PROGRAM SafetyInterface_MtrCntrl051
VAR
	
	pMtrRunning: POINTER TO ConvMtrRunningPuck;
	pSafety: POINTER TO Plc2PlcDataSafetyPuckConv;
	
// Stn051_05_StnMain.MotorCtrl
// Call to motor control function block for each main line motor	
// Blue Return - Enc52:  5,6  Enc53: 3,4,5,6
// Red Return  - Enc52:  3,4   Enc53:2
// Grn Return  - Enc52: 1,2   Enc53: 1
//  Blu receive bypass - Enc52: 7
	{attribute 'TcLinkToOSO':= '	
		.Enc052Mtr01.iDisconnectOk :=  <0,1,3>TIIB[N16S00 (AL1332)]^N16S03 (AL2341)^TxPDO^input byte 3;
		.Enc052Mtr02.iDisconnectOk :=  <0,1,3>TIIB[N16S00 (AL1332)]^N16S07 (AL2341)^TxPDO^input byte 1;
		.Enc052Mtr03.iDisconnectOk :=  <0,1,4>TIIB[N16S00 (AL1332)]^N16S03 (AL2341)^TxPDO^input byte 1;
		.Enc052Mtr04.iDisconnectOk :=  <0,1,3>TIIB[N16S00 (AL1332)]^N16S07 (AL2341)^TxPDO^input byte 3;
		.Enc052Mtr05.iDisconnectOk :=  <0,1,4>TIIB[N16S00 (AL1332)]^N16S03 (AL2341)^TxPDO^input byte 3;
		.Enc052Mtr06.iDisconnectOk :=  <0,1,4>TIIB[N16S00 (AL1332)]^N16S07 (AL2341)^TxPDO^input byte 1;
		.Enc052Mtr07.iDisconnectOk :=  <0,1,4>TIIB[N16S00 (AL1332)]^N16S07 (AL2341)^TxPDO^input byte 3;
		.Enc053Mtr01.iDisconnectOk :=  <0,1,2>TIIB[N21S00 (AL1332)]^N21S01 (AL2341)^TxPDO^input byte 3;
		.Enc053Mtr02.iDisconnectOk :=  <0,1,3>TIIB[N21S00 (AL1332)]^N21S01 (AL2341)^TxPDO^input byte 1;
		.Enc053Mtr03.iDisconnectOk :=  <0,1,3>TIIB[N21S00 (AL1332)]^N21S01 (AL2341)^TxPDO^input byte 1;
		.Enc053Mtr04.iDisconnectOk :=  <0,1,3>TIIB[N21S00 (AL1332)]^N21S01 (AL2341)^TxPDO^input byte 1;
		.Enc053Mtr05.iDisconnectOk :=  <0,1,4>TIIB[N24S00 (AL1332)]^N24S05 (AL2341)^TxPDO^input byte 3;
		.Enc053Mtr06.iDisconnectOk :=  <0,1,3>TIIB[N21S00 (AL1332)]^N21S01 (AL2341)^TxPDO^input byte 1'}
	{attribute 'TcLinkTo':= '	
		.Enc052Mtr01.iOverloadTripped := TIIB[N15S06 (EL1008)]^Channel 6^Input;
		.Enc052Mtr02.iOverloadTripped := TIIB[N15S06 (EL1008)]^Channel 8^Input;
		.Enc052Mtr03.iOverloadTripped := TIIB[N15S07 (EL1008)]^Channel 2^Input;
		.Enc052Mtr04.iOverloadTripped := TIIB[N15S07 (EL1008)]^Channel 4^Input;
		.Enc052Mtr05.iOverloadTripped := TIIB[N15S07 (EL1008)]^Channel 6^Input;
		.Enc052Mtr06.iOverloadTripped := TIIB[N15S07 (EL1008)]^Channel 8^Input;
		.Enc052Mtr07.iOverloadTripped := TIIB[N15S08 (EL1008)]^Channel 2^Input;
		.Enc053Mtr01.iOverloadTripped := TIIB[N20S06 (EL1008)]^Channel 6^Input;
		.Enc053Mtr02.iOverloadTripped := TIIB[N20S06 (EL1008)]^Channel 8^Input;
		.Enc053Mtr03.iOverloadTripped := TIIB[N20S07 (EL1008)]^Channel 2^Input;
		.Enc053Mtr04.iOverloadTripped := TIIB[N20S07 (EL1008)]^Channel 4^Input;
		.Enc053Mtr05.iOverloadTripped := TIIB[N20S07 (EL1008)]^Channel 6^Input;
		.Enc053Mtr06.iOverloadTripped := TIIB[N20S07 (EL1008)]^Channel 8^Input;
		.Enc052Mtr01.iRunning := TIIB[N15S06 (EL1008)]^Channel 5^Input;
		.Enc052Mtr02.iRunning := TIIB[N15S06 (EL1008)]^Channel 7^Input;
		.Enc052Mtr03.iRunning := TIIB[N15S07 (EL1008)]^Channel 1^Input;
		.Enc052Mtr04.iRunning := TIIB[N15S07 (EL1008)]^Channel 3^Input;
		.Enc052Mtr05.iRunning := TIIB[N15S07 (EL1008)]^Channel 5^Input;
		.Enc052Mtr06.iRunning := TIIB[N15S07 (EL1008)]^Channel 7^Input;
		.Enc052Mtr07.iRunning := TIIB[N15S08 (EL1008)]^Channel 1^Input;
		.Enc053Mtr01.iRunning := TIIB[N20S06 (EL1008)]^Channel 5^Input;
		.Enc053Mtr02.iRunning := TIIB[N20S06 (EL1008)]^Channel 7^Input;
		.Enc053Mtr03.iRunning := TIIB[N20S07 (EL1008)]^Channel 1^Input;
		.Enc053Mtr04.iRunning := TIIB[N20S07 (EL1008)]^Channel 3^Input;
		.Enc053Mtr05.iRunning := TIIB[N20S07 (EL1008)]^Channel 5^Input;
		.Enc053Mtr06.iRunning := TIIB[N20S07 (EL1008)]^Channel 7^Input;
		.Enc052Mtr01.oRun := TIIB[N15S12 (EL2008)]^Channel 5^Output;
		.Enc052Mtr02.oRun := TIIB[N15S12 (EL2008)]^Channel 6^Output;
		.Enc052Mtr03.oRun := TIIB[N15S12 (EL2008)]^Channel 7^Output;
		.Enc052Mtr04.oRun := TIIB[N15S12 (EL2008)]^Channel 8^Output;
		.Enc052Mtr05.oRun := TIIB[N15S13 (EL2008)]^Channel 1^Output;
		.Enc052Mtr06.oRun := TIIB[N15S13 (EL2008)]^Channel 2^Output;
		.Enc052Mtr07.oRun := TIIB[N15S13 (EL2008)]^Channel 3^Output;
		.Enc053Mtr01.oRun := TIIB[N20S12 (EL2008)]^Channel 4^Output;
		.Enc053Mtr02.oRun := TIIB[N20S12 (EL2008)]^Channel 5^Output;
		.Enc053Mtr03.oRun := TIIB[N20S12 (EL2008)]^Channel 6^Output;
		.Enc053Mtr04.oRun := TIIB[N20S12 (EL2008)]^Channel 7^Output;
		.Enc053Mtr05.oRun := TIIB[N20S12 (EL2008)]^Channel 8^Output;
		.Enc053Mtr06.oRun := TIIB[N20S13 (EL2008)]^Channel 1^Output'}
	MtrCtrls: ConvMtrCtrlsPuck;

	MtrNOKtoRun : BOOL;	  	//not used at this time, see the attached action for details.
	cntMotorStartIndex: DINT;	
	tmrMotorStartIndex: TON;


END_VAR
VAR CONSTANT	
	
	cMaxMotorStartIndex :DINT := 9;  //If starting pairs of motors  adjust to max number of motors "per enclosure" /2
	
END_VAR

pMtrRunning := ADR(gProduced_SafetyInterfaceConv.MtrRunning);
pSafety := ADR(gProduced_SafetyInterfaceConv);

//Create sequenced motor start index - to prevent inrush overloads at time of motor start		
tmrMotorStartIndex(IN:=NOT tmrMotorStartIndex.Q,PT:=T#300ms);		
IF tmrMotorStartIndex.Q THEN 		
	cntMotorStartIndex := cntMotorStartIndex + 1;	
	IF cntMotorStartIndex > cMaxMotorStartIndex THEN 	
		cntMotorStartIndex := 1;
	END_IF	
END_IF		

// Call action code block that does call for each main line motor		
MotorCtrl();

//distibute the incoming stn data (consumed data from stn) to single produced outgoing to all stns
//MEMCPY(ADR(gProduced_SafetyInterfaceConv.gMtrRunningStn051), ADR(gMtrRunning), SizeOf(gProduced_SafetyInterfaceConv.gMtrRunningStn051));

ACTION MotorCtrl:
// Stn051_05_StnMain.MotorCtrl
// Call to motor control function block for each main line motor	
// Blue Return - Enc52:  5,6  Enc53: 3,4,5,6
// Red Return  - Enc52:  3,4   Enc53:2
// Grn Return  - Enc52: 1,2   Enc53: 1
//  Blu receive bypass - Enc52: 7

MtrCtrls.Enc052Mtr01(	
	CycleAuto := gConsumed_Stn051ToSafetyInterface.CycleAuto,
	CycleReset := gConsumed_Stn051ToSafetyInterface.CycleReset,
	NOKtoRun := pSafety^.Enc052.iEstopRlyTripped,	
//	NOKtoRun := pSafety^.Enc052.iEstopRlyTripped OR 
//		NOT gConsumed_Stn051ToSafetyInterface.Stn051PLCData[2].3 OR 
//		NOT gConsumed_Stn051ToSafetyInterface_OK,		
	StartIndexThisMotor := 1,
	StartIndexCurrent := cntMotorStartIndex,
	hoMtrName := 'Enc052-Mtr1',
	MtrRunning => pMtrRunning^.Enc052Mtr01);

MtrCtrls.Enc052Mtr02(	
	CycleAuto := gConsumed_Stn051ToSafetyInterface.CycleAuto,
	CycleReset := gConsumed_Stn051ToSafetyInterface.CycleReset,
	NOKtoRun := pSafety^.Enc052.iEstopRlyTripped,	
//	NOKtoRun := pSafety^.Enc052.iEstopRlyTripped OR 
//		NOT gConsumed_Stn051ToSafetyInterface.Stn051PLCData[2].3 OR 
//		NOT gConsumed_Stn051ToSafetyInterface_OK,		
	StartIndexThisMotor := 1,
	StartIndexCurrent := cntMotorStartIndex,
	hoMtrName := 'Enc052-Mtr2',
	MtrRunning => pMtrRunning^.Enc052Mtr02);

MtrCtrls.Enc052Mtr03(	
	CycleAuto := gConsumed_Stn051ToSafetyInterface.CycleAuto,
	CycleReset := gConsumed_Stn051ToSafetyInterface.CycleReset,
	NOKtoRun := pSafety^.Enc052.iEstopRlyTripped,	
//	NOKtoRun := pSafety^.Enc052.iEstopRlyTripped OR 
//		NOT gConsumed_Stn051ToSafetyInterface.Stn051PLCData[2].3 OR 
//		NOT gConsumed_Stn051ToSafetyInterface_OK,		
	StartIndexThisMotor := 2,
	StartIndexCurrent := cntMotorStartIndex,
	hoMtrName := 'Enc052-Mtr3',
	MtrRunning => pMtrRunning^.Enc052Mtr03);

MtrCtrls.Enc052Mtr04(	
	CycleAuto := gConsumed_Stn051ToSafetyInterface.CycleAuto,
	CycleReset := gConsumed_Stn051ToSafetyInterface.CycleReset,
	NOKtoRun := pSafety^.Enc052.iEstopRlyTripped,	
//	NOKtoRun := pSafety^.Enc052.iEstopRlyTripped OR 
//		NOT gConsumed_Stn051ToSafetyInterface.Stn051PLCData[2].3 OR 
//		NOT gConsumed_Stn051ToSafetyInterface_OK,		
	StartIndexThisMotor := 2,
	StartIndexCurrent := cntMotorStartIndex,
	hoMtrName := 'Enc052-Mtr4',
	MtrRunning => pMtrRunning^.Enc052Mtr04);

MtrCtrls.Enc052Mtr05(	
	CycleAuto := gConsumed_Stn051ToSafetyInterface.CycleAuto,
	CycleReset := gConsumed_Stn051ToSafetyInterface.CycleReset,
	NOKtoRun := pSafety^.Enc052.iEstopRlyTripped,	
//	NOKtoRun := pSafety^.Enc052.iEstopRlyTripped OR 
//		NOT gConsumed_Stn051ToSafetyInterface.Stn051PLCData[2].3 OR 
//		NOT gConsumed_Stn051ToSafetyInterface_OK,		
	StartIndexThisMotor := 3,
	StartIndexCurrent := cntMotorStartIndex,
	hoMtrName := 'Enc052-Mtr5',
	MtrRunning => pMtrRunning^.Enc052Mtr05);

MtrCtrls.Enc052Mtr06(	
	CycleAuto := gConsumed_Stn051ToSafetyInterface.CycleAuto,
	CycleReset := gConsumed_Stn051ToSafetyInterface.CycleReset,
	NOKtoRun := pSafety^.Enc052.iEstopRlyTripped,	
//	NOKtoRun := pSafety^.Enc052.iEstopRlyTripped OR 
//		NOT gConsumed_Stn051ToSafetyInterface.Stn051PLCData[2].3 OR 
//		NOT gConsumed_Stn051ToSafetyInterface_OK,		
	StartIndexThisMotor := 3,
	StartIndexCurrent := cntMotorStartIndex,
	hoMtrName := 'Enc052-Mtr6',
	MtrRunning => pMtrRunning^.Enc052Mtr06);

MtrCtrls.Enc052Mtr07(	
	CycleAuto := gConsumed_Stn051ToSafetyInterface.CycleAuto,
	CycleReset := gConsumed_Stn051ToSafetyInterface.CycleReset,
	NOKtoRun := pSafety^.Enc052.iEstopRlyTripped,	
//	NOKtoRun := pSafety^.Enc052.iEstopRlyTripped OR 
//		NOT gConsumed_Stn051ToSafetyInterface.Stn051PLCData[2].3 OR 
//		NOT gConsumed_Stn051ToSafetyInterface_OK,		
	StartIndexThisMotor := 4,
	StartIndexCurrent := cntMotorStartIndex,
	hoMtrName := 'Enc052-Mtr7',
	MtrRunning => pMtrRunning^.Enc052Mtr07);

MtrCtrls.Enc053Mtr01(	
	CycleAuto := gConsumed_Stn051ToSafetyInterface.CycleAuto,
	CycleReset := gConsumed_Stn051ToSafetyInterface.CycleReset,
	NOKtoRun := pSafety^.Enc053.iEstopRlyTripped,	
//	NOKtoRun := pSafety^.Enc053.iEstopRlyTripped OR 
//		NOT gConsumed_Stn051ToSafetyInterface.Stn051PLCData[2].3 OR 
//		NOT gConsumed_Stn051ToSafetyInterface_OK,		
	StartIndexThisMotor := 1,
	StartIndexCurrent := cntMotorStartIndex,
	hoMtrName := 'Enc053-Mtr1',
	MtrRunning => pMtrRunning^.Enc053Mtr01);

MtrCtrls.Enc053Mtr02(	
	CycleAuto := gConsumed_Stn051ToSafetyInterface.CycleAuto,
	CycleReset := gConsumed_Stn051ToSafetyInterface.CycleReset,
	NOKtoRun := pSafety^.Enc053.iEstopRlyTripped,	
//	NOKtoRun := pSafety^.Enc053.iEstopRlyTripped OR 
//		NOT gConsumed_Stn051ToSafetyInterface.Stn051PLCData[2].3 OR 
//		NOT gConsumed_Stn051ToSafetyInterface_OK,		
	StartIndexThisMotor := 1,
	StartIndexCurrent := cntMotorStartIndex,
	hoMtrName := 'Enc053-Mtr2',
	MtrRunning => pMtrRunning^.Enc053Mtr02);

MtrCtrls.Enc053Mtr03(	
	CycleAuto := gConsumed_Stn051ToSafetyInterface.CycleAuto,
	CycleReset := gConsumed_Stn051ToSafetyInterface.CycleReset,
	NOKtoRun := pSafety^.Enc053.iEstopRlyTripped,	
//	NOKtoRun := pSafety^.Enc053.iEstopRlyTripped OR 
//		NOT gConsumed_Stn051ToSafetyInterface.Stn051PLCData[2].3 OR 
//		NOT gConsumed_Stn051ToSafetyInterface_OK,		
	StartIndexThisMotor := 2,
	StartIndexCurrent := cntMotorStartIndex,
	hoMtrName := 'Enc053-Mtr3',
	MtrRunning => pMtrRunning^.Enc053Mtr03);

MtrCtrls.Enc053Mtr04(	
	CycleAuto := gConsumed_Stn051ToSafetyInterface.CycleAuto,
	CycleReset := gConsumed_Stn051ToSafetyInterface.CycleReset,
	NOKtoRun := pSafety^.Enc053.iEstopRlyTripped,	
//	NOKtoRun := pSafety^.Enc053.iEstopRlyTripped OR 
//		NOT gConsumed_Stn051ToSafetyInterface.Stn051PLCData[2].3 OR 
//		NOT gConsumed_Stn051ToSafetyInterface_OK,		
	StartIndexThisMotor := 2,
	StartIndexCurrent := cntMotorStartIndex,
	hoMtrName := 'Enc053-Mtr4',
	MtrRunning => pMtrRunning^.Enc053Mtr04);

MtrCtrls.Enc053Mtr05(	
	CycleAuto := gConsumed_Stn051ToSafetyInterface.CycleAuto,
	CycleReset := gConsumed_Stn051ToSafetyInterface.CycleReset,
	NOKtoRun := pSafety^.Enc053.iEstopRlyTripped,	
//	NOKtoRun := pSafety^.Enc053.iEstopRlyTripped OR 
//		NOT gConsumed_Stn051ToSafetyInterface.Stn051PLCData[2].3 OR 
//		NOT gConsumed_Stn051ToSafetyInterface_OK,		
	StartIndexThisMotor := 3,
	StartIndexCurrent := cntMotorStartIndex,
	hoMtrName := 'Enc053-Mtr5',
	MtrRunning => pMtrRunning^.Enc053Mtr05);

MtrCtrls.Enc053Mtr06(	
	CycleAuto := gConsumed_Stn051ToSafetyInterface.CycleAuto,
	CycleReset := gConsumed_Stn051ToSafetyInterface.CycleReset,
	NOKtoRun := pSafety^.Enc053.iEstopRlyTripped,	
//	NOKtoRun := pSafety^.Enc053.iEstopRlyTripped OR 
//		NOT gConsumed_Stn051ToSafetyInterface.Stn051PLCData[2].3 OR 
//		NOT gConsumed_Stn051ToSafetyInterface_OK,		
	StartIndexThisMotor := 3,
	StartIndexCurrent := cntMotorStartIndex,
	hoMtrName := 'Enc053-Mtr6',
	MtrRunning => pMtrRunning^.Enc053Mtr06);
	
//For each motor that the station needs running information but NOT actually controlling the output… 
//(populate the running bit from the produced consumed logic)

// Populate motor running for motors controlled (outputs linked) by other stations
//gMtrRunning.Enc062Mtr07 := gConsumed_Stn901To902.ScratchPad[10].0;
END_ACTION

END_PROGRAM

(* stored: Version 1.1.0.1, ProductVersion 3.1.4024.6
   POU SafetyInterface_MtrCntrl051: Id {10c89f34-e83e-40f6-8da5-3c17679cd46d}, SpecialFunc None
   Action MotorCtrl: Id {25a6197f-86ab-4eba-9db2-3b52f4792434} *)
